FUNCTION_BLOCK FB_AnalogDeviceRampControl
VAR
	i : INT;
END_VAR

(*MFC*)
FOR i:=1 TO 12 DO
	IF GVL_IO.aMaxValueController[i] <> 0 THEN
		GVL_IO.aAnalogOutputIO[i] := LREAL_TO_INT(GVL_IO.aController[i].rControlValue); //Write to Device
		GVL_IO.aController_PV[i] := (GVL_IO.aAnalogInputIO[i] / GVL_CONSTANT.EL3064MaxValueH) * GVL_IO.aMaxValueController[i];
		GVL_IO.aController_CV[i] := LREAL_TO_REAL((GVL_IO.aController[i].rControlValue / GVL_CONSTANT.EL3064MaxValueH)*GVL_IO.aMaxValueController[i]);
		GVL_IO.aController[i]();
	END_IF
END_FOR


(*EPC*)
FOR i:=20 TO 23 DO
	IF GVL_IO.aMaxValueController[i] <> 0 THEN
		GVL_IO.aAnalogOutputIO[i] := LREAL_TO_INT(GVL_IO.aController[i].rControlValue); //Write to Device
		GVL_IO.aController_PV[i] := (GVL_IO.aAnalogInputIO[i] / GVL_CONSTANT.EL3064MaxValueH) * GVL_IO.aMaxValueController[i];
		GVL_IO.aController_CV[i] := LREAL_TO_REAL((GVL_IO.aController[i].rControlValue / GVL_CONSTANT.EL3064MaxValueH)*GVL_IO.aMaxValueController[i]);
		GVL_IO.aController[i]();
	END_IF
END_FOR


IF ( GVL_IO.aController_CV[27] > 10 ) THEN
	GVL_IO.aDigitalOutputIO[2].0 := TRUE;
ELSE
	GVL_IO.aDigitalOutputIO[2].0 := FALSE;
END_IF

//jhkang aController 의 Input은 언제 들어감?
//Temp Controller
GVL_IO.temperatureTV := REAL_TO_INT(GVL_IO.aController[E_aAnalogInputIO_Index.E_PV_Susceptor_Temp].input.targetValue);
GVL_IO.wE3508_CV := LREAL_TO_WORD(GVL_IO.aController[E_aAnalogInputIO_Index.E_PV_Susceptor_Temp].rControlValue); //Write to Temperature Controller
GVL_IO.aController_PV[E_aAnalogInputIO_Index.E_PV_Susceptor_Temp] := WORD_TO_REAL(GVL_IO.wE3508_PV);
GVL_IO.aController_CV[E_aAnalogInputIO_Index.E_PV_Susceptor_Temp] := WORD_TO_REAL(GVL_IO.wE3508_CV);
GVL_IO.aController[E_aAnalogInputIO_Index.E_PV_Susceptor_Temp]();

//Temp Pressure Controller
GVL_IO.pressureTV := REAL_TO_INT(GVL_IO.aController[E_aAnalogInputIO_Index.E_PV_Reactor_Pressure].input.targetValue);				
GVL_IO.wIqPlus_CV := LREAL_TO_WORD(GVL_IO.aController[E_aAnalogInputIO_Index.E_PV_Reactor_Pressure].rControlValue); //Write to Pressure Controller
GVL_IO.aController_PV[E_aAnalogInputIO_Index.E_PV_Reactor_Pressure] := WORD_TO_REAL(GVL_IO.wIqPlus_CDG2_PV);
GVL_IO.aController_CV[E_aAnalogInputIO_Index.E_PV_Reactor_Pressure] := WORD_TO_REAL(GVL_IO.wIqPlus_CV);
GVL_IO.aController[E_aAnalogInputIO_Index.E_PV_Reactor_Pressure]();

//Rotation Controller
GVL_IO.rotationTV := REAL_TO_INT(GVL_IO.aController[E_aAnalogInputIO_Index.E_PV_susceptorRotation].input.targetValue);			
GVL_IO.rRotation_ControlValue := LREAL_TO_REAL(GVL_IO.aController[E_aAnalogInputIO_Index.E_PV_susceptorRotation].rControlValue); //Write to Rotation Controller (rpm)
GVL_IO.aController_PV[E_aAnalogInputIO_Index.E_PV_susceptorRotation] := GVL_IO.nRotation_Converted_PV;
GVL_IO.aController_CV[E_aAnalogInputIO_Index.E_PV_susceptorRotation] := GVL_IO.rRotation_ControlValue;
GVL_IO.aController[E_aAnalogInputIO_Index.E_PV_susceptorRotation]();

END_FUNCTION_BLOCK

(* stored: Version 1.1.0.1, ProductVersion 3.1.4024.15
   POU FB_AnalogDeviceRampControl: Id {901ef948-d319-4e50-9c34-c06b07342954}, SpecialFunc None *)
